Universal Robots PolyScope program: Museum.urp

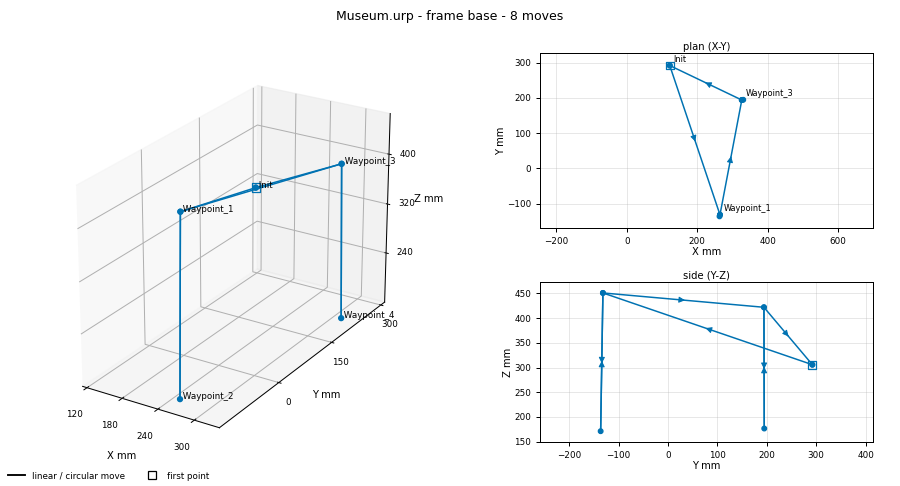
[picture p0: tool path of Museum.urp in frame base, 8 of 8 moves have a stored position in this frame; points joined in program order, loops and branches not executed]
Program Museum (installation=default directory=/programs/Mursal createdIn=5.11.11.1010533 lastSavedIn=5.11.11.1010533 robotSerialNumber=20205300864)
Calibrated DH parameters: a=[-0.000166, -0.243494, -0.153108, 0.000057, -0.000123, 0]; d=[0.151897, -1.34267, 53.988124, -52.514559, 0.085283, 0.092193]; alpha=[1.572472, -0.003756, 0.002824, 1.570807, -1.572621, 0]; deltaTheta=[0, 0.020704, 7.033215, -0.770746, 0.000004, 0]
Robot Program (runOnlyOnce=true)
  MoveL speed 250 mm/s, acceleration 1200 mm/s^2 (useActiveTCP=true) feature=Base
    Waypoint Init: TCP in base x=122.118 y=292.121 z=305.736 mm, rx=1.1346 ry=-2.9295 rz=0 rad; joints [91.64, -87.587, -91.765, -90.542, 90.034, 859.399] deg
    Waypoint Waypoint_1: TCP in base x=264.738 y=-131.613 z=450.872 mm, rx=0.0016 ry=-3.1415 rz=-0.0001 rad; joints [-0.127, -96.409, -39.239, -134.252, 89.89, 809.868] deg
    Waypoint Waypoint_2: TCP in base x=263.462 y=-136.186 z=171.15 mm, rx=0.0016 ry=-3.1415 rz=-0.0002 rad; joints [-1.294, -93.122, -125.108, -51.672, 90.066, 808.848] deg
    URCap Gripper (Robotiq_Grippers, Robotiq Inc.) dataModel(position=100.0, force=1.0, speed=100.0, positionInDouble=100.0, forceInDouble=1.0, speedInDouble=100.0, slaveIds=[9], blocking=true, robotCompliant=false)
    Waypoint Waypoint_1: TCP in base x=264.738 y=-131.613 z=450.872 mm, rx=0.0016 ry=-3.1415 rz=-0.0001 rad; joints [-0.127, -96.409, -39.239, -134.252, 89.89, 809.868] deg
    Waypoint Waypoint_3: TCP in base x=326.691 y=194.178 z=421.861 mm, rx=0.0288 ry=-3.1413 rz=-0.0001 rad; joints [50.937, -119.588, -15.527, -134.784, 89.812, 859.915] deg
    Waypoint Waypoint_4: TCP in base x=330.819 y=194.821 z=176.582 mm, rx=-0.0065 ry=3.1416 rz=0 rad; joints [50.308, -112.214, -98.425, -59.255, 89.983, 860.234] deg
    URCap Gripper (Robotiq_Grippers, Robotiq Inc.) dataModel(position=0.0, force=1.0, speed=100.0, positionInDouble=0.0, forceInDouble=1.0, speedInDouble=100.0, slaveIds=[9], blocking=true, robotCompliant=false)
    Waypoint Waypoint_3: TCP in base x=326.691 y=194.178 z=421.861 mm, rx=0.0288 ry=-3.1413 rz=-0.0001 rad; joints [50.937, -119.588, -15.527, -134.784, 89.812, 859.915] deg
    Waypoint Init: TCP in base x=122.118 y=292.121 z=305.736 mm, rx=1.1346 ry=-2.9295 rz=0 rad; joints [91.64, -87.587, -91.765, -90.542, 90.034, 859.399] deg
